{attribute addProperty BoxType "EP9224-0037-0017"}
{attribute addProperty Id "Error_UsBIT10.1251Error_UpBIT10.1252Warning_UsBIT10.1253Warning_UpBIT10.1254Status_UsBIT10.1255Status_UpBIT10.1256Channel_ErrorBIT10.1257Error_Sum_CurrentBIT10.1258Warning_Sum_CurrentBIT10.1259TxPDO_StateBIT10.12515TxPDO_ToggleBIT10.12516"}
{attribute addProperty CRC "2723206043"}
{attribute addProperty SizeInBites "16"}
{attribute addProperty SizeInBytes "2"}
TYPE Status_A250D39B :
STRUCT
	{attribute addProperty Name "Error_Us"}
	Error_Us : BIT;
	{attribute addProperty Name "Error_Up"}
	Error_Up : BIT;
	{attribute addProperty Name "Warning_Us"}
	Warning_Us : BIT;
	{attribute addProperty Name "Warning_Up"}
	Warning_Up : BIT;
	{attribute addProperty Name "Status_Us"}
	Status_Us : BIT;
	{attribute addProperty Name "Status_Up"}
	Status_Up : BIT;
	{attribute addProperty Name "Channel_Error"}
	Channel_Error : BIT;
	{attribute addProperty Name "Error_Sum_Current"}
	Error_Sum_Current : BIT;
	{attribute addProperty Name "Warning_Sum_Current"}
	Warning_Sum_Current : BIT;
	{attribute 'hide'}
	reserve_1_BIT_0 : BIT;
	{attribute 'hide'}
	reserve_1_BIT_1 : BIT;
	{attribute 'hide'}
	reserve_1_BIT_2 : BIT;
	{attribute 'hide'}
	reserve_1_BIT_3 : BIT;
	{attribute 'hide'}
	reserve_1_BIT_4 : BIT;
	{attribute addProperty Name "TxPDO_State"}
	TxPDO_State : BIT;
	{attribute addProperty Name "TxPDO_Toggle"}
	TxPDO_Toggle : BIT;
END_STRUCT
END_TYPE

(* stored: Version 1.2.0.0, ProductVersion 3.1.4024.9
   DUT Status_A250D39B: Id {6cb651a7-a2c4-4964-9a36-294c5c776eeb} *)
